SYSTEM WORKER_HMI_1 (* System Configuration *)
  (* Standard: 61499-1 *)
  (* Version 0.3, 2003-12-05, JHC, Rockwell Automation, Renamed from NEWSYSTEM. *)
  (* Version 0.2, 2002-11-05, JHC, Rockwell Automation, Fixed missing (empty) FBD in Application. *)
  (* Version 0.1, 2002-01-17, JHC, Rockwell Automation, Minor cleanup *)
  (* Version 0.0, 2000-05-27, JHC, Rockwell Automation *)
  APPLICATION APP1
  END_APPLICATION
  DEVICE WORKER_HMI_DEVICE : FRAME_DEVICE(BOUNDS := [1100,300,600,400], GRID := [1,1])
    RESOURCE WORKER_HMI_PROCESSOR : PANEL_RESOURCE(ROWS := 6, COLS := 2)
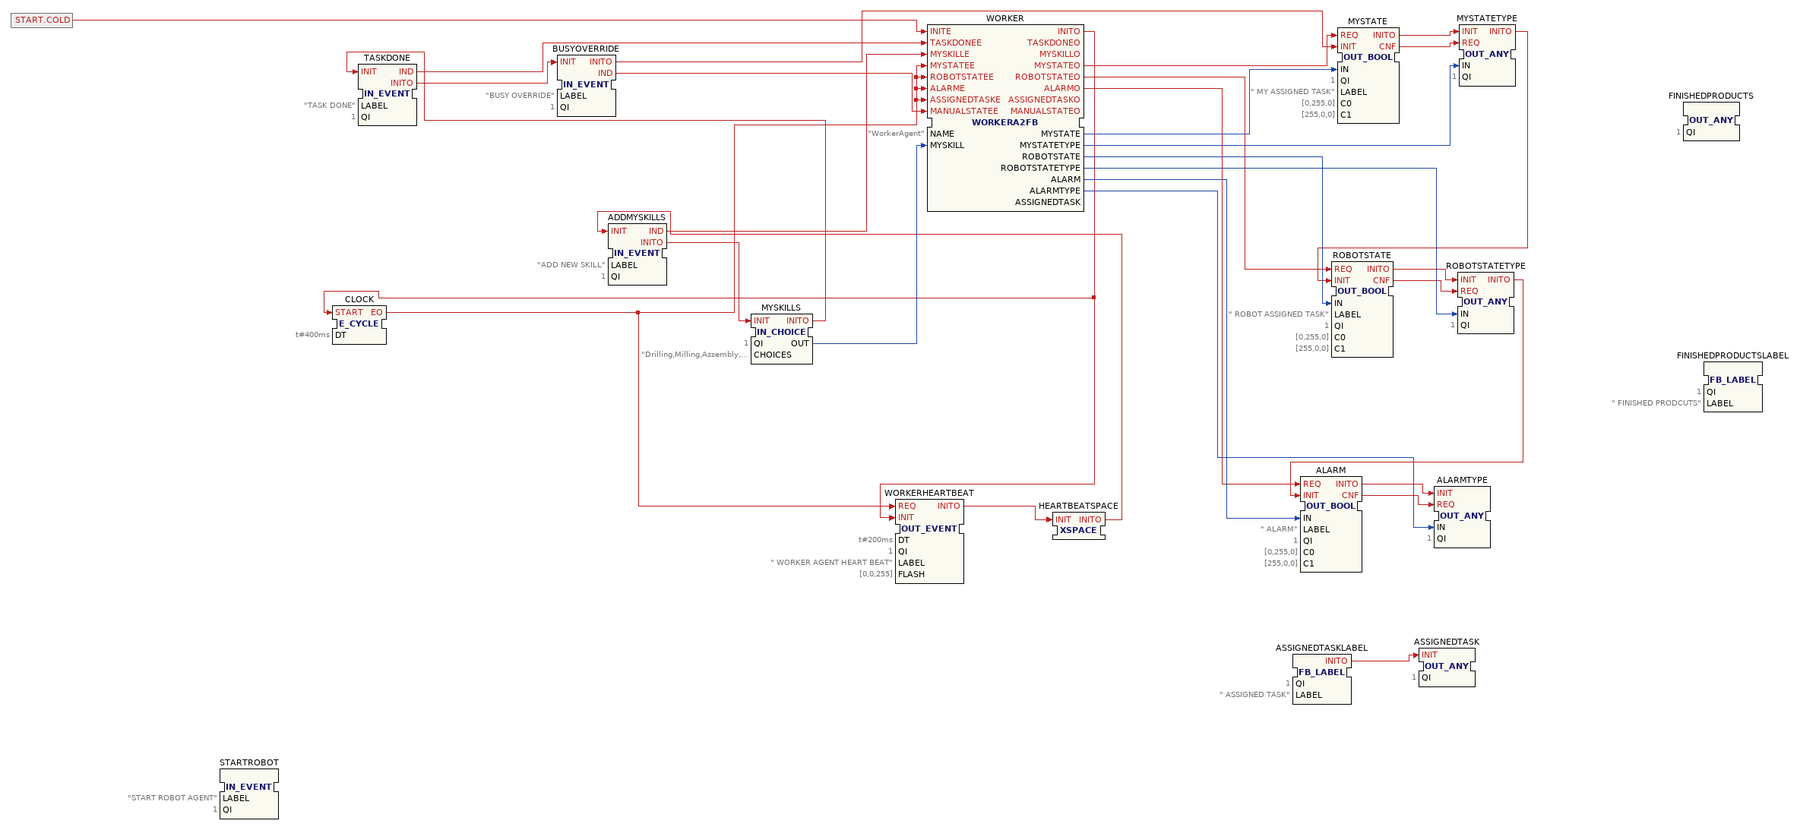
      FBS
        WORKER : WORKERA2FB(NAME := "WorkerAgent");
        MYSTATETYPE : OUT_ANY(QI := 1);
        ALARMTYPE : OUT_ANY(QI := 1);
        ALARM : OUT_BOOL(LABEL := "                                    ALARM", QI := 1, C0 := [0,255,0], C1 := [255,0,0]);
        ASSIGNEDTASKLABEL : FB_LABEL(QI := 1, LABEL := "                                   ASSIGNED TASK");
        ASSIGNEDTASK : OUT_ANY(QI := 1);
        FINISHEDPRODUCTSLABEL : FB_LABEL(QI := 1, LABEL := "                               FINISHED PRODCUTS");
        FINISHEDPRODUCTS : OUT_ANY(QI := 1);
        ROBOTSTATETYPE : OUT_ANY(QI := 1);
        STARTROBOT : IN_EVENT(LABEL := "START ROBOT AGENT", QI := 1);
        BUSYOVERRIDE : IN_EVENT(LABEL := "BUSY OVERRIDE", QI := 1);
        ADDMYSKILLS : IN_EVENT(LABEL := "ADD NEW SKILL", QI := 1);
        MYSKILLS : IN_CHOICE(QI := 1, CHOICES := "Drilling,Milling,Assembly,Painting,Shaping");
        WORKERHEARTBEAT : OUT_EVENT(DT := t#200ms, QI := 1, LABEL := "                         WORKER AGENT HEART BEAT", FLASH := [0,0,255]);
        CLOCK : E_CYCLE(DT := t#400ms);
        HEARTBEATSPACE : XSPACE;
        TASKDONE : IN_EVENT(LABEL := "TASK DONE", QI := 1);
        MYSTATE : OUT_BOOL(QI := 1, LABEL := "                               MY ASSIGNED TASK", C0 := [0,255,0], C1 := [255,0,0]);
        ROBOTSTATE : OUT_BOOL(LABEL := "                            ROBOT ASSIGNED TASK", QI := 1, C0 := [0,255,0], C1 := [255,0,0]);
      END_FBS
      EVENT_CONNECTIONS
        ALARM.INITO TO ALARMTYPE.INIT;
        ALARM.CNF TO ALARMTYPE.REQ;
        ADDMYSKILLS.IND TO WORKER.MYSKILLE;
        ADDMYSKILLS.INITO TO MYSKILLS.INIT;
        CLOCK.EO TO WORKER.MYSTATEE;
        CLOCK.EO TO WORKER.ROBOTSTATEE;
        CLOCK.EO TO WORKER.ALARME;
        CLOCK.EO TO WORKER.ASSIGNEDTASKE;
        CLOCK.EO TO WORKERHEARTBEAT.REQ;
        TASKDONE.IND TO WORKER.TASKDONEE;
        MYSTATE.INITO TO MYSTATETYPE.INIT;
        MYSTATE.CNF TO MYSTATETYPE.REQ;
        ROBOTSTATE.INITO TO ROBOTSTATETYPE.INIT;
        ROBOTSTATE.CNF TO ROBOTSTATETYPE.REQ;
        WORKER.MYSTATEO TO MYSTATE.REQ;
        WORKER.ROBOTSTATEO TO ROBOTSTATE.REQ;
        WORKER.ALARMO TO ALARM.REQ;
        ASSIGNEDTASKLABEL.INITO TO ASSIGNEDTASK.INIT;
        START.COLD TO WORKER.INITE;
        WORKER.INITO TO WORKERHEARTBEAT.INIT;
        WORKERHEARTBEAT.INITO TO HEARTBEATSPACE.INIT;
        HEARTBEATSPACE.INITO TO ADDMYSKILLS.INIT;
        MYSKILLS.INITO TO TASKDONE.INIT;
        TASKDONE.INITO TO BUSYOVERRIDE.INIT;
        BUSYOVERRIDE.INITO TO MYSTATE.INIT;
        MYSTATETYPE.INITO TO ROBOTSTATE.INIT;
        ROBOTSTATETYPE.INITO TO ALARM.INIT;
        BUSYOVERRIDE.IND TO WORKER.MANUALSTATEE;
        WORKER.INITO TO CLOCK.START;
      END_CONNECTIONS
      DATA_CONNECTIONS
        MYSKILLS.OUT TO WORKER.MYSKILL;
        WORKER.MYSTATE TO MYSTATE.IN;
        WORKER.ROBOTSTATE TO ROBOTSTATE.IN;
        WORKER.MYSTATETYPE TO MYSTATETYPE.IN;
        WORKER.ROBOTSTATETYPE TO ROBOTSTATETYPE.IN;
        WORKER.ALARM TO ALARM.IN;
        WORKER.ALARMTYPE TO ALARMTYPE.IN;
      END_CONNECTIONS
    END_RESOURCE
  END_DEVICE
END_SYSTEM
